# B&R Automation Studio project SimulationsBoard
Automation Studio 4.7.2.98; Das ist mein Einfuehrungsprojekt zum Simboard

## Configuration Config1

CPU X20CP1584, AutomationRuntime C4.72, Build 4.1.2, Vc V4.72.0

### Task classes (Cpu.sw)
```
Cyclic#4:
  Aufgabe_7 <- Aufgabe_7.prg
Binaries: udbdef, FWRules, TCData, iomap, ashwac, Role, sysconf, arconfig, asfw, User, ashwd
Libraries: standard
```

### Hardware
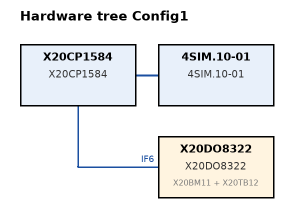
```
4SIM.10-01 : 4SIM.10-01 v1.3.0.0  [PLK1 -> X20CP1584.IF3 [Cable Type=PowerlinkCable, Length=10, Version=1.0.0.2]]
X20BM11 : X20BM11 v1.0.0.1  [X2X1 -> X20CP1584.IF6]
X20CP1584 : X20CP1584 v1.6.0.0
  Connector IF2:
    ActivateDevice = 1
    Mode = Manual
    InternetAddress = 10.36.37.14
    SubnetMask = 255.255.255.0
X20DO8322 : X20DO8322 v1.1.0.0  [SS1 -> X20TB12.SS; SL -> X20BM11.SL1]
X20TB12 : X20TB12 v1.0.0.0
```

### IoMap.iom - X20CP1584/IoMap.iom
```iecst
VAR_CONFIG
	::switch_left AT %IX."4SIM.10-01".DigitalInput01;
	::switch_right AT %IX."4SIM.10-01".DigitalInput02;
	::LED1_red AT %QX."4SIM.10-01".DigitalOutput03;
	::LED1_orange AT %QX."4SIM.10-01".DigitalOutput04;
	::LED1_green AT %QX."4SIM.10-01".DigitalOutput05;
	::LED2_red AT %QX."4SIM.10-01".DigitalOutput06;
	::LED2_orange AT %QX."4SIM.10-01".DigitalOutput07;
	::LED2_green AT %QX."4SIM.10-01".DigitalOutput08;
	::LED3_red AT %QX."4SIM.10-01".DigitalOutput09;
	::LED3_orange AT %QX."4SIM.10-01".DigitalOutput10;
	::LED3_green AT %QX."4SIM.10-01".DigitalOutput11;
	::LED4_red AT %QX."4SIM.10-01".DigitalOutput12;
	::LED4_orange AT %QX."4SIM.10-01".DigitalOutput13;
	::LED4_green AT %QX."4SIM.10-01".DigitalOutput14;
	::seven_seg AT %QW."4SIM.10-01".AnalogOutput01;
	::but_1 AT %IX."4SIM.10-01".DigitalInput03;
	::but_2 AT %IX."4SIM.10-01".DigitalInput04;
	::but_3 AT %IX."4SIM.10-01".DigitalInput05;
	::but_4 AT %IX."4SIM.10-01".DigitalInput06;
	::pot_1 AT %IW."4SIM.10-01".AnalogInput01;
	::pot_2 AT %IW."4SIM.10-01".AnalogInput02;
	::takt AT %IW."4SIM.10-01".Encoder01;
	::LED_SW_left AT %QX."4SIM.10-01".DigitalOutput01;
	::LED_SW_right AT %QX."4SIM.10-01".DigitalOutput02;
END_VAR
```

## Logical view

### Global.typ - Global data types
```iecst
TYPE
	LED_stat : 	STRUCT
		off : BOOL;
		pressed : BOOL;
		long_pressed : BOOL;
		time : UDINT;
	END_STRUCT;
END_TYPE
```

### Global.var - Global variables
```iecst
VAR
	switch_left : BOOL;
	switch_right : BOOL;
	but_1 : BOOL;
	but_3 : BOOL;
	but_2 : BOOL;
	but_4 : BOOL;
END_VAR
(*LEDS*)
VAR
	LED1_green : BOOL;
	LED1_red : BOOL;
	LED1_orange : BOOL;
END_VAR
(*Insert your comment here.*)
VAR
	LED2_green : BOOL;
	LED2_red : BOOL;
	LED2_orange : BOOL;
END_VAR
(*Insert your comment here.*)
VAR
	LED3_green : BOOL;
	LED3_red : BOOL;
	LED3_orange : BOOL;
END_VAR
(*Insert your comment here.*)
VAR
	LED4_green : BOOL;
	LED4_red : BOOL;
	LED4_orange : BOOL;
	LED_SW_left : BOOL;
	LED_SW_right : BOOL;
END_VAR
(*Analog*)
VAR
	pot_1 : INT;
	pot_2 : INT;
	takt : UINT;
	seven_seg : INT;
END_VAR
```

### Program Logical/Aufgabe_1 (ANSIC)

#### Init.c
```c
#include <bur/plctypes.h>

#ifdef _DEFAULT_INCLUDES
	#include <AsDefault.h>
#endif

void _INIT ProgramInit(void)
{
	switch_left	=0;
	switch_right = 0;
	but_1 = 0;
	but_3 = 0;
	but_2 = 0;
	but_4 = 0;

	LED1_green = 0;
	LED1_red = 0;
	LED1_orange = 0;

	LED2_green = 0;
	LED2_red = 0;
	LED2_orange = 0;

	LED3_green = 0;
	LED3_red = 0;
	LED3_orange = 0;

	LED4_green = 0;
	LED4_red = 0;
	LED4_orange = 0;

	pot_1 = 0;
	pot_2 = 0;
	takt = 0;
	seven_seg = 420;

}
```

### Program Logical/Aufgabe_2 (ANSIC)

#### Variables.var
```iecst
VAR
	R_TRIG_BUT_1 : R_TRIG;
	R_TRIG_BUT_2 : R_TRIG;
	R_TRIG_BUT_3 : R_TRIG;
	R_TRIG_BUT_4 : R_TRIG;
	R_TRIG_SW : R_TRIG;
	F_TRIG_SW : F_TRIG;
END_VAR
```

#### Cyclic.c
```c
#include <bur/plctypes.h>
#include <standard.h>       /* prototypes for STANDARD-Library */
#ifdef _DEFAULT_INCLUDES
	#include <AsDefault.h>
#endif

void _CYCLIC ProgramCyclic(void)
{
	R_TRIG_BUT_1.CLK = but_1;
	R_TRIG_BUT_2.CLK = but_2;
	R_TRIG_BUT_3.CLK = but_3;
	R_TRIG_BUT_4.CLK = but_4;
	R_TRIG_SW.CLK = switch_left;
	F_TRIG_SW.CLK = switch_left;

	R_TRIG(&R_TRIG_BUT_1);
	R_TRIG(&R_TRIG_BUT_2);
	R_TRIG(&R_TRIG_BUT_3);
	R_TRIG(&R_TRIG_BUT_4);
	R_TRIG(&R_TRIG_SW);
	F_TRIG(&F_TRIG_SW);

	if(F_TRIG_SW.Q)
	{
		LED1_red = 0;
		LED1_green = 0;
		LED2_red = 0;
		LED2_green = 0;
		LED3_red = 0;
		LED3_green = 0;
		LED4_red = 0;
		LED4_green = 0;
	}

	if(R_TRIG_SW.Q)
	{
		LED1_red = 1;
		LED1_green = 0;
		LED2_red = 1;
		LED2_green = 0;
		LED3_red = 1;
		LED3_green = 0;
		LED4_red = 1;
		LED4_green = 0;
	}

	if(R_TRIG_BUT_1.Q)
	{
		if(LED1_red != 0 || LED1_green !=0)
		{
			LED1_red = !LED1_red;
			LED1_green = !LED1_green;
		}
	}
	if(R_TRIG_BUT_2.Q)
	{
		if(LED2_red != 0 || LED2_green !=0)
		{
			LED2_red = !LED2_red;
			LED2_green = !LED2_green;
		}
	}
	if(R_TRIG_BUT_3.Q)
	{
		if(LED3_red != 0 || LED3_green !=0)
		{
			LED3_red = !LED3_red;
			LED3_green = !LED3_green;
		}
	}
	if(R_TRIG_BUT_4.Q)
	{
		if(LED4_red != 0 || LED4_green !=0)
		{
			LED4_red = !LED4_red;
			LED4_green = !LED4_green;
		}
	}

	LED_SW_left = switch_left;
}
```

#### Init.c
```c
#include <bur/plctypes.h>

#ifdef _DEFAULT_INCLUDES
#include <AsDefault.h>
#endif

void _INIT ProgramInit(void)
{
	switch_left	=0;
	switch_right = 0;
	but_1 = 0;
	but_3 = 0;
	but_2 = 0;
	but_4 = 0;

	LED1_green = 0;
	LED1_red = 0;
	LED1_orange = 0;

	LED2_green = 0;
	LED2_red = 0;
	LED2_orange = 0;

	LED3_green = 0;
	LED3_red = 0;
	LED3_orange = 0;

	LED4_green = 0;
	LED4_red = 0;
	LED4_orange = 0;

	pot_1 = 0;
	pot_2 = 0;
	takt = 0;
	seven_seg = 420;
}
```

### Program Logical/Aufgabe_3 (ANSIC)

#### Variables.var
```iecst
VAR
	R_TRIG_BUT_1 : R_TRIG;
	TON_BUT_1 : TON;
	R_TRIG_BUT_2 : R_TRIG;
	TON_BUT_2 : TON;
	R_TRIG_BUT_3 : R_TRIG;
	TON_BUT_3 : TON;
	R_TRIG_BUT_4 : R_TRIG;
	TON_BUT_4 : TON;
	R_TRIG_SW : R_TRIG;
	F_TRIG_SW : F_TRIG;
END_VAR
```

#### Cyclic.c
```c
#include <bur/plctypes.h>
#include <standard.h>       /* prototypes for STANDARD-Library */
#ifdef _DEFAULT_INCLUDES
#include <AsDefault.h>
#endif

void handleButton(R_TRIGtyp* edge, TONtyp* timer,BOOL* but, BOOL* red, BOOL* green)
{
	edge->CLK = timer->Q;
	timer->PT = 3000;
	timer->IN = *but;
	TON(timer);
	R_TRIG(edge);

	if(edge->Q)
	{
		if(*red != 0 || *green !=0)
		{
			*red = !*red;
			*green = !*green;
		}
	}
}

void _CYCLIC ProgramCyclic(void)
{
	handleButton(&R_TRIG_BUT_1, &TON_BUT_1, &but_1, &LED1_red, &LED1_green);
	handleButton(&R_TRIG_BUT_2, &TON_BUT_2, &but_2, &LED2_red, &LED2_green);
	handleButton(&R_TRIG_BUT_3, &TON_BUT_3, &but_3, &LED3_red, &LED3_green);
	handleButton(&R_TRIG_BUT_4, &TON_BUT_4, &but_4, &LED4_red, &LED4_green);

	R_TRIG_SW.CLK = switch_left;
	F_TRIG_SW.CLK = switch_left;

	R_TRIG(&R_TRIG_SW);
	F_TRIG(&F_TRIG_SW);

	if(F_TRIG_SW.Q)
	{
		LED1_red = 0;
		LED1_green = 0;
		LED2_red = 0;
		LED2_green = 0;
		LED3_red = 0;
		LED3_green = 0;
		LED4_red = 0;
		LED4_green = 0;
	}

	if(R_TRIG_SW.Q)
	{
		LED1_red = 1;
		LED1_green = 0;
		LED2_red = 1;
		LED2_green = 0;
		LED3_red = 1;
		LED3_green = 0;
		LED4_red = 1;
		LED4_green = 0;
	}
	LED_SW_left = switch_left;
}
```

### Program Logical/Aufgabe_4 (ANSIC)

#### Cyclic.c
```c
#include <bur/plctypes.h>

#ifdef _DEFAULT_INCLUDES
	#include <AsDefault.h>
#endif

void _CYCLIC ProgramCyclic(void)
{
	if(switch_left)
	{
		seven_seg = (100*pot_1/32767);
	}
	else
	{
		seven_seg = 0;
	}
	LED_SW_left = switch_left;
}
```

#### Init.c
```c
#include <bur/plctypes.h>

#ifdef _DEFAULT_INCLUDES
#include <AsDefault.h>
#endif

void _INIT ProgramInit(void)
{
	switch_left	=0;
	switch_right = 0;
	but_1 = 0;
	but_3 = 0;
	but_2 = 0;
	but_4 = 0;

	LED1_green = 0;
	LED1_red = 0;
	LED1_orange = 0;

	LED2_green = 0;
	LED2_red = 0;
	LED2_orange = 0;

	LED3_green = 0;
	LED3_red = 0;
	LED3_orange = 0;

	LED4_green = 0;
	LED4_red = 0;
	LED4_orange = 0;

	pot_1 = 0;
	pot_2 = 0;
	takt = 0;
	seven_seg = 420;
}
```

### Program Logical/Aufgabe_5 (ANSIC)

#### Cyclic.c
```c
#include <bur/plctypes.h>

#ifdef _DEFAULT_INCLUDES
	#include <AsDefault.h>
#endif

int add(int, int);
int subtract(int, int);
int multiply(int, int);
int divide(int, int);
void handleButton(R_TRIGtyp* , BOOL* , int (*fun)(int, int), int, int, int*);

void _CYCLIC ProgramCyclic(void)
{
	handleButton(&R_TRIG_BUT_1, &but_1, add, savedVal_Pot_1,savedVal_Pot_2, &seven_seg);
	handleButton(&R_TRIG_BUT_2, &but_2, subtract, savedVal_Pot_1,savedVal_Pot_2, &seven_seg);
	handleButton(&R_TRIG_BUT_3, &but_3, multiply, savedVal_Pot_1,savedVal_Pot_2, &seven_seg);
	handleButton(&R_TRIG_BUT_4, &but_4, divide, savedVal_Pot_1,savedVal_Pot_2, &seven_seg);

	F_TRIG_SW.CLK = switch_left;
	F_TRIG_SW_RIGHT.CLK = switch_right;

	//Anzeige linkes Poti
	if(switch_left && !switch_right)
		seven_seg = (100*pot_1/32767);
	//anzeige rechtes Poti
	if(!switch_left && switch_right)
		seven_seg = (100*pot_2/32767);

	//Wenn beide ein sind: --- anzeigen
	if(switch_left && switch_right)
		seven_seg = 1000;

	if(F_TRIG_SW.Q)
		savedVal_Pot_1 = 100*pot_1/32767;
	if(F_TRIG_SW_RIGHT.Q)
		savedVal_Pot_2 = 100*pot_2/32767;

	F_TRIG(&F_TRIG_SW);
	F_TRIG(&F_TRIG_SW_RIGHT);

	LED_SW_left = switch_left;
	LED_SW_right = switch_right;
}

int add(int a, int b )
{
	return a+b;
}
int subtract(int a, int b )
{
	return a-b;
}

int multiply(int a, int b )
{
	return a*b;
}
int divide(int a, int b )
{
	return a/b;
}

void handleButton(R_TRIGtyp* edge, BOOL* but, int (*fun)(int, int), int a, int b, int* output)
{
	edge->CLK = *but;
	R_TRIG(edge);

	if(edge->Q)
		*output = fun(a,b);
}
```

### Program Logical/Aufgabe_6 (ANSIC)

#### Cyclic.c
```c
#include <bur/plctypes.h>

#ifdef _DEFAULT_INCLUDES
	#include <AsDefault.h>
#endif

void _CYCLIC ProgramCyclic(void)
{
	R_TRIG_SW.CLK = switch_left;
	F_TRIG_SW.CLK = switch_left;

	R_TRIG(&R_TRIG_SW);
	F_TRIG(&F_TRIG_SW);

	if(F_TRIG_SW.Q)
	{
		LED1_red = 0;
		LED1_green = 0;
	}

	if(R_TRIG_SW.Q)
	{
		LED1_red = 1;
		LED1_green = 0;
	}

	if(switch_left)
	{
		LED1_red = !LED1_red;
		LED1_green = !LED1_green;
	}
	LED_SW_left = switch_left;
}
```

### Program Logical/Aufgabe_7 (ANSIC)

#### Variables.var
```iecst
VAR
	R_TRIG_BUT_1 : R_TRIG;
	TON_BUT_1 : TON;
	R_TRIG_BUT_2 : R_TRIG;
	TON_BUT_2 : TON;
	R_TRIG_BUT_3 : R_TRIG;
	TON_BUT_3 : TON;
	R_TRIG_BUT_4 : R_TRIG;
	TON_BUT_4 : TON;
	R_TRIG_SW : R_TRIG;
	F_TRIG_SW : F_TRIG;
	F_TRIG_SW_RIGHT : F_TRIG;
	savedVal_Pot_1 : USINT;
	savedVal_Pot_2 : USINT;
END_VAR
```

#### Cyclic.c
```c
#include <bur/plctypes.h>

#ifdef _DEFAULT_INCLUDES
	#include <AsDefault.h>
#endif

void _CYCLIC ProgramCyclic(void)
{
	R_TRIG_SW.CLK = switch_left;
	F_TRIG_SW.CLK = switch_left;

	R_TRIG(&R_TRIG_SW);
	F_TRIG(&F_TRIG_SW);

	if(F_TRIG_SW.Q)
	{
		LED1_orange = 0;
		LED2_orange = 0;
		LED3_orange = 0;
		LED4_orange = 0;
	}

	if(R_TRIG_SW.Q)
	{
		LED1_orange = 1;
		LED2_orange = 1;
		LED3_orange = 1;
		LED4_orange = 1;
	}

	LED_SW_left = switch_left;
}
```

#### Init.c
```c
#include <bur/plctypes.h>

#ifdef _DEFAULT_INCLUDES
#include <AsDefault.h>
#endif

void _INIT ProgramInit(void)
{
	switch_left	=0;
	switch_right = 0;

	but_1 = 0;
	but_3 = 0;
	but_2 = 0;
	but_4 = 0;

	LED1_green = 0;
	LED1_red = 0;
	LED1_orange = 0;

	LED2_green = 0;
	LED2_red = 0;
	LED2_orange = 0;

	LED3_green = 0;
	LED3_red = 0;
	LED3_orange = 0;

	LED4_green = 0;
	LED4_red = 0;
	LED4_orange = 0;

	pot_1 = 0;
	pot_2 = 0;
	takt = 0;
	seven_seg = 00;
}
```

Listed in the project but not available here: Logical/Libraries
